# EPICS autosave request: iocBoot/ioc13bmd_aerotech/auto_settings.req
file "CARS_motor_settings.req",         P=$(P), M=m113
file "CARS_motor_settings.req",         P=$(P), M=m114
file "CARS_motor_settings.req",         P=$(P), M=m115
file "CARS_motor_settings.req",         P=$(P), M=m116
file "CARS_motor_settings.req",         P=$(P), M=m117
file "CARS_motor_settings.req",         P=$(P), M=m118
file "CARS_motor_settings.req",         P=$(P), M=m119
